FUNCTION_BLOCK PUBL_2 (* Two-Variable Local Group Publisher *)
  (* Standard: 61499-1; Classification: Communications; Function: 2-variable local group publisher *)
  (* Version 0.1, 2002-05-02, JHC, Rockwell Automation, Optimized. *)
  (* Version 0.0, 2001-10-02, JHC, Rockwell Automation, Copied/modified from PUBLISH_2 *)
  (* Compiler header: package fb.rt.net; *)
  (* Compiler Java IBM VisualAge 3.0 *)
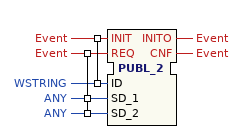
  EVENT_INPUT
    INIT WITH ID; (* Service Initialization *)
    REQ WITH SD_1, SD_2; (* Service Request *)
  END_EVENT
  EVENT_OUTPUT
    INITO; (* Initialization Confirm *)
    CNF; (* Service Confirmation *)
  END_EVENT
  VAR_INPUT
    ID : WSTRING; (* Local Group Name-Default is FB Instance Name *)
    SD_1 : ANY; (* Data to Send *)
    SD_2 : ANY; (* Data to Send *)
  END_VAR
END_FUNCTION_BLOCK
